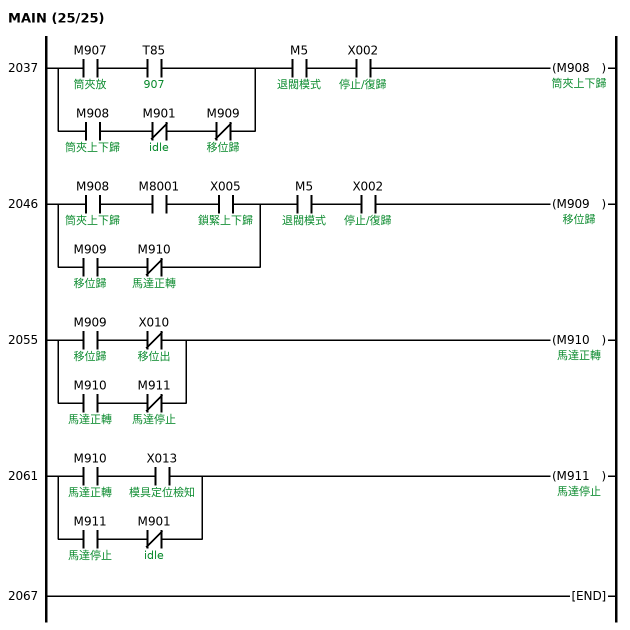
[picture p24: ladder of MAIN, rungs at steps 2037 to 2067]
2037  LD      M907  ; 筒夾放
      AND     T85  ; 907
      LD      M908  ; 筒夾上下歸
      ANI     M901  ; idle
      ANI     M909  ; 移位歸
      ORB
      AND     M5  ; 退閥模式
      AND     X002  ; 停止/復歸
      OUT     M908  ; 筒夾上下歸
2046  LD      M908  ; 筒夾上下歸
      AND     M8001
      AND     X005  ; 鎖緊上下歸
      LD      M909  ; 移位歸
      ANI     M910  ; 馬達正轉
      ORB
      AND     M5  ; 退閥模式
      AND     X002  ; 停止/復歸
      OUT     M909  ; 移位歸
2055  LD      M909  ; 移位歸
      ANI     X010  ; 移位出
      LD      M910  ; 馬達正轉
      ANI     M911  ; 馬達停止
      ORB
      OUT     M910  ; 馬達正轉
2061  LD      M910  ; 馬達正轉
      AND     X013  ; 模具定位檢知
      LD      M911  ; 馬達停止
      ANI     M901  ; idle
      ORB
      OUT     M911  ; 馬達停止
2067  END
END_PROGRAM

// device comments not shown above
M6  ; 退閥啟動
M502  ; 筒夾放鬆PB
M505  ; 夾緊氣缸放PB
M511  ; 伺服異常重置PB
M580  ; power on
M581  ; idle
M582  ; 移位出
M583  ; 筒夾上下出
M584  ; 伺服起動
M585  ; 伺服停止
M586  ; 筒夾放
M587  ; 筒夾上下歸
M588  ; 移位歸
D723  ; **************
D778  ; D776/10
R201  ; ******
R240  ; type1轉距補償(輸出)
R241  ; type2轉距補償(輸出)
R260  ; 手動速度(設定)
R261  ; 手動轉距(設定)
R270  ; 點膠速度(設定)
R304  ; DA轉距m
R305  ; DA轉距n
R380  ; type1轉距上限(輸出)
R381  ; type1轉距下限(輸出)
R382  ; type2轉距上限(輸出)
R383  ; type2轉距下限(輸出)
R404  ; DA速度m
R405  ; DA速度n
R1000  ; #1著座速度(set)
R1002  ; #1鎖緊速度(set)
R1004  ; #1著座扭力(set)
R1006  ; #1鎖緊扭力(set)
R1008  ; #1扭力上限(set)
R1010  ; #1扭力下限(set)
R1012  ; #1扭力補償(set)
R1020  ; #1著座速度(output)
R1022  ; #1鎖緊速度(output)
R1024  ; #1著座扭力(output)
R1026  ; #1鎖緊扭力(output)
R1028  ; #1扭力上限(output)
R1030  ; #1扭力下限(output)
R1032  ; #1扭力補償(output)
R1034  ; #1扭力上限+補償
R1036  ; #1扭力下限+補償
R1040  ; #2著座速度(set)
R1042  ; #2鎖緊速度(set)
R1044  ; #2著座扭力(set)
R1046  ; #2鎖緊扭力(set)
R1048  ; #2扭力上限(set)
R1050  ; #2扭力下限(set)
R1052  ; #2扭力補償(set)
R1060  ; #2著座速度(output)
R1062  ; #2鎖緊速度(output)
R1064  ; #2著座扭力(output)
R1066  ; #2鎖緊扭力(output)
R1068  ; #2扭力上限(output)
R1070  ; #2扭力下限(output)
R1072  ; #2扭力補償(output)
R1074  ; #2扭力上限+補償
R1076  ; #2扭力下限+補償
R1080  ; #3著座速度(set)
R1082  ; #3鎖緊速度(set)
R1084  ; #3著座扭力(set)
R1086  ; #3鎖緊扭力(set)
R1088  ; #3扭力上限(set)
R1090  ; #3扭力下限(set)
R1092  ; #3扭力補償(set)
R1100  ; #3著座速度(output)
R1102  ; #3鎖緊速度(output)
R1104  ; #3著座扭力(output)
R1106  ; #3鎖緊扭力(output)
R1108  ; #3扭力上限(output)
R1110  ; #3扭力下限(output)
R1112  ; #3扭力補償(output)
R1114  ; #3扭力上限+補償
R1116  ; #3扭力下限+補償
R1120  ; #4著座速度(set)
R1122  ; #4鎖緊速度(set)
R1124  ; #4著座扭力(set)
R1126  ; #4鎖緊扭力(set)
R1128  ; #4扭力上限(set)
R1130  ; #4扭力下限(set)
R1132  ; #4扭力補償(set)
R1140  ; #4著座速度(output)
R1142  ; #4鎖緊速度(output)
R1144  ; #4著座扭力(output)
R1146  ; #4鎖緊扭力(output)
R1148  ; #4扭力上限(output)
R1150  ; #4扭力下限(output)
R1152  ; #4扭力補償(output)
R1154  ; #4扭力上限+補償
R1156  ; #4扭力下限+補償
R1160  ; #5著座速度(set)
R1162  ; #5鎖緊速度(set)
R1164  ; #5著座扭力(set)
R1166  ; #5鎖緊扭力(set)
R1168  ; #5扭力上限(set)
R1170  ; #5扭力下限(set)
R1172  ; #5扭力補償(set)
R1180  ; #5著座速度(output)
R1182  ; #5鎖緊速度(output)
R1184  ; #5著座扭力(output)
R1186  ; #5鎖緊扭力(output)
R1188  ; #5扭力上限(output)
R1190  ; #5扭力下限(output)
R1192  ; #5扭力補償(output)
R1194  ; #5扭力上限+補償
R1196  ; #5扭力下限+補償
R1200  ; #6著座速度(set)
R1202  ; #6鎖緊速度(set)
R1204  ; #6著座扭力(set)
R1206  ; #6鎖緊扭力(set)
R1208  ; #6扭力上限(set)
R1210  ; #6扭力下限(set)
R1212  ; #6扭力補償(set)
R1220  ; #6著座速度(output)
R1222  ; #6鎖緊速度(output)
R1224  ; #6著座扭力(output)
R1226  ; #6鎖緊扭力(output)
R1228  ; #6扭力上限(output)
R1230  ; #6扭力下限(output)
R1232  ; #6扭力補償(output)
R1234  ; #6扭力上限+補償
R1236  ; #6扭力下限+補償
R1240  ; #7著座速度(set)
R1242  ; #7鎖緊速度(set)
R1244  ; #7著座扭力(set)
R1246  ; #7鎖緊扭力(set)
R1248  ; #7扭力上限(set)
R1250  ; #7扭力下限(set)
R1252  ; #7扭力補償(set)
R1260  ; #7著座速度(output)
R1262  ; #7鎖緊速度(output)
R1264  ; #7著座扭力(output)
R1266  ; #7鎖緊扭力(output)
R1268  ; #7扭力上限(output)
R1270  ; #7扭力下限(output)
R1272  ; #7扭力補償(output)
R1274  ; #7扭力上限+補償
R1276  ; #7扭力下限+補償
R1280  ; #8著座速度(set)
R1282  ; #8鎖緊速度(set)
R1284  ; #8著座扭力(set)
R1286  ; #8鎖緊扭力(set)
R1288  ; #8扭力上限(set)
R1290  ; #8扭力下限(set)
R1292  ; #8扭力補償(set)
R1300  ; #8著座速度(output)
R1302  ; #8鎖緊速度(output)
R1304  ; #8著座扭力(output)
R1306  ; #8鎖緊扭力(output)
R1308  ; #8扭力上限(output)
R1310  ; #8扭力下限(output)
R1312  ; #8扭力補償(output)
R1314  ; #8扭力上限+補償
R1316  ; #8扭力下限+補償
R1320  ; #9著座速度(set)
R1322  ; #9鎖緊速度(set)
R1324  ; #9著座扭力(set)
R1326  ; #9鎖緊扭力(set)
R1328  ; #9扭力上限(set)
R1330  ; #9扭力下限(set)
R1332  ; #9扭力補償(set)
R1340  ; #9著座速度(output)
R1342  ; #9鎖緊速度(output)
R1344  ; #9著座扭力(output)
R1346  ; #9鎖緊扭力(output)
R1348  ; #9扭力上限(output)
R1350  ; #9扭力下限(output)
R1352  ; #9扭力補償(output)
R1354  ; #9扭力上限+補償
R1356  ; #9扭力下限+補償
R1360  ; #10著座速度(set)
R1362  ; #10鎖緊速度(set)
R1364  ; #10著座扭力(set)
R1366  ; #10鎖緊扭力(set)
R1368  ; #10扭力上限(set)
R1370  ; #10扭力下限(set)
R1372  ; #10扭力補償(set)
R1380  ; #10著座速度(output)
R1382  ; #10鎖緊速度(output)
R1384  ; #10著座扭力(output)
R1386  ; #10鎖緊扭力(output)
R1388  ; #10扭力上限(output)
R1390  ; #10扭力下限(output)
R1392  ; #10扭力補償(output)
R1394  ; #10扭力上限+補償
R1396  ; #10扭力下限+補償
T2  ; 筒夾放鬆sol
T5  ; 夾緊氣缸放sol
